# EPICS autosave request: iocs/hamamatsuIOC/iocBoot/iocHamamatsu/auto_settings.req
file "hamamatsu_settings.req",      P=$(P),  R=cam1:
file "NDStdArrays_settings.req",    P=$(P),  R=image1:
file "commonPlugin_settings.req",   P=$(P)
